% RSLogix 500 project P2_BAK007.RSS, saved by version 8.30.00.16 %
PROJECT "UNTITLED"    % processor: Bul.1763 MicroLogix 1100 Series B %

PROGRAM FILES
  LAD 2 "MAIN"  4 rungs
  LAD 3 "I/O"  8 rungs
  LAD 4 "CONTROLS"  6 rungs
  LAD 5 "CYCLE"  5 rungs

DATA FILES
  O0 OUTPUT  4 elements
  I1 INPUT  6 elements
  S2 STATUS  66 elements
  B3 BINARY  6 elements
  T4 TIMER  1 elements
  C5 COUNTER  1 elements
  R6 CONTROL  1 elements
  N7 INTEGER  1 elements
  F8 FLOAT  1 elements

LADDER 2 "MAIN"
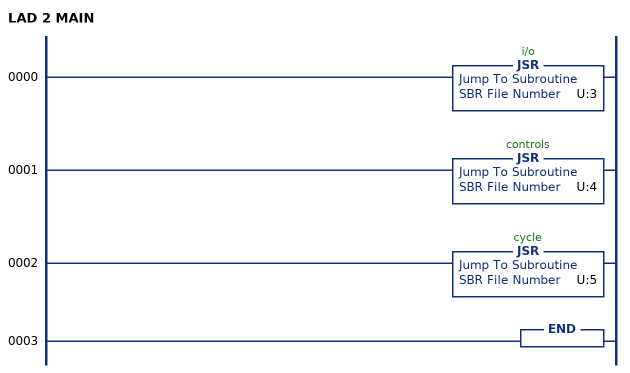
% Rung: 0 %
SOR JSR U:3 EOR
%   U:3  "i/o" %
% Rung: 1 %
SOR JSR U:4 EOR
%   U:4  "controls" %
% Rung: 2 %
SOR JSR U:5 EOR
%   U:5  "cycle" %
% Rung: 3 %
SOR END EOR

LADDER 3 "I/O"
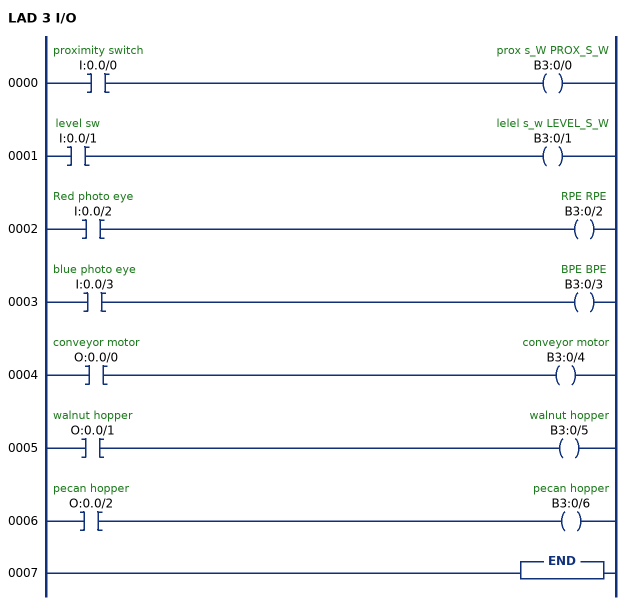
% Rung: 0 %
SOR XIC I:0.0/0 OTE B3:0/0 EOR
%   I:0.0/0  "proximity switch" %
%   B3:0/0  PROX_S_W  "prox s_W" %
% Rung: 1 %
SOR XIC I:0.0/1 OTE B3:0/1 EOR
%   I:0.0/1  "level sw" %
%   B3:0/1  LEVEL_S_W  "lelel s_w" %
% Rung: 2 %
SOR XIC I:0.0/2 OTE B3:0/2 EOR
%   I:0.0/2  "Red photo eye" %
%   B3:0/2  RPE  "RPE" %
% Rung: 3 %
SOR XIC I:0.0/3 OTE B3:0/3 EOR
%   I:0.0/3  "blue photo eye" %
%   B3:0/3  BPE  "BPE" %
% Rung: 4 %
SOR XIC O:0.0/0 OTE B3:0/4 EOR
%   O:0.0/0  "conveyor motor" %
%   B3:0/4  "conveyor motor" %
% Rung: 5 %
SOR XIC O:0.0/1 OTE B3:0/5 EOR
%   O:0.0/1  "walnut hopper" %
%   B3:0/5  "walnut hopper" %
% Rung: 6 %
SOR XIC O:0.0/2 OTE B3:0/6 EOR
%   O:0.0/2  "pecan hopper" %
%   B3:0/6  "pecan hopper" %
% Rung: 7 %
SOR END EOR

LADDER 4 "CONTROLS"
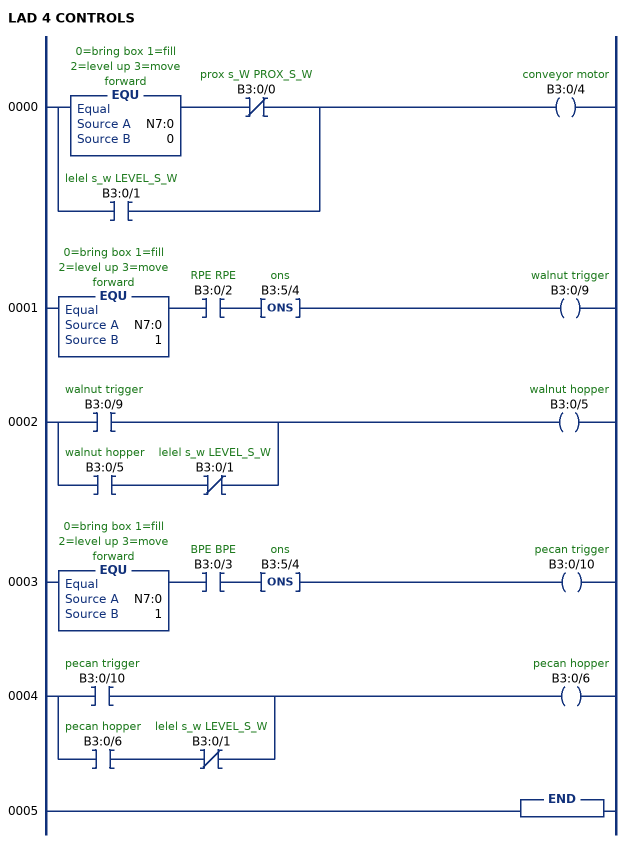
% Rung: 0 %
SOR BST EQU N7:0 0 XIO B3:0/0 NXB XIC B3:0/1 BND OTE B3:0/4 EOR
%   N7:0  "0=bring box 1=fill 2=level up 3=move forward" %
%   B3:0/0  PROX_S_W  "prox s_W" %
%   B3:0/1  LEVEL_S_W  "lelel s_w" %
%   B3:0/4  "conveyor motor" %
% Rung: 1 %
SOR EQU N7:0 1 XIC B3:0/2 ONS B3:5/4 OTE B3:0/9 EOR
%   N7:0  "0=bring box 1=fill 2=level up 3=move forward" %
%   B3:0/2  RPE  "RPE" %
%   B3:5/4  "ons" %
%   B3:0/9  "walnut trigger" %
% Rung: 2 %
SOR BST XIC B3:0/9 NXB XIC B3:0/5 XIO B3:0/1 BND OTE B3:0/5 EOR
%   B3:0/9  "walnut trigger" %
%   B3:0/5  "walnut hopper" %
%   B3:0/1  LEVEL_S_W  "lelel s_w" %
% Rung: 3 %
SOR EQU N7:0 1 XIC B3:0/3 ONS B3:5/4 OTE B3:0/10 EOR
%   N7:0  "0=bring box 1=fill 2=level up 3=move forward" %
%   B3:0/3  BPE  "BPE" %
%   B3:5/4  "ons" %
%   B3:0/10  "pecan trigger" %
% Rung: 4 %
SOR BST XIC B3:0/10 NXB XIC B3:0/6 XIO B3:0/1 BND OTE B3:0/6 EOR
%   B3:0/10  "pecan trigger" %
%   B3:0/6  "pecan hopper" %
%   B3:0/1  LEVEL_S_W  "lelel s_w" %
% Rung: 5 %
SOR END EOR

LADDER 5 "CYCLE"
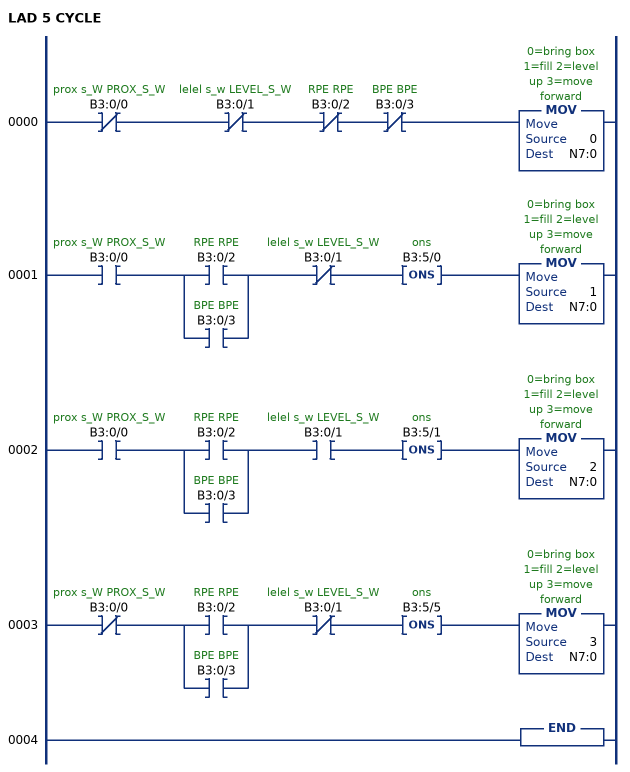
% Rung: 0 %
SOR XIO B3:0/0 XIO B3:0/1 XIO B3:0/2 XIO B3:0/3 MOV 0 N7:0 EOR
%   B3:0/0  PROX_S_W  "prox s_W" %
%   B3:0/1  LEVEL_S_W  "lelel s_w" %
%   B3:0/2  RPE  "RPE" %
%   B3:0/3  BPE  "BPE" %
%   N7:0  "0=bring box 1=fill 2=level up 3=move forward" %
% Rung: 1 %
SOR XIC B3:0/0 BST XIC B3:0/2 NXB XIC B3:0/3 BND XIO B3:0/1 ONS B3:5/0 MOV 1 N7:0 EOR
%   B3:0/0  PROX_S_W  "prox s_W" %
%   B3:0/2  RPE  "RPE" %
%   B3:0/3  BPE  "BPE" %
%   B3:0/1  LEVEL_S_W  "lelel s_w" %
%   B3:5/0  "ons" %
%   N7:0  "0=bring box 1=fill 2=level up 3=move forward" %
% Rung: 2 %
SOR XIC B3:0/0 BST XIC B3:0/2 NXB XIC B3:0/3 BND XIC B3:0/1 ONS B3:5/1 MOV 2 N7:0 EOR
%   B3:0/0  PROX_S_W  "prox s_W" %
%   B3:0/2  RPE  "RPE" %
%   B3:0/3  BPE  "BPE" %
%   B3:0/1  LEVEL_S_W  "lelel s_w" %
%   B3:5/1  "ons" %
%   N7:0  "0=bring box 1=fill 2=level up 3=move forward" %
% Rung: 3 %
SOR XIO B3:0/0 BST XIC B3:0/2 NXB XIC B3:0/3 BND XIO B3:0/1 ONS B3:5/5 MOV 3 N7:0 EOR
%   B3:0/0  PROX_S_W  "prox s_W" %
%   B3:0/2  RPE  "RPE" %
%   B3:0/3  BPE  "BPE" %
%   B3:0/1  LEVEL_S_W  "lelel s_w" %
%   B3:5/5  "ons" %
%   N7:0  "0=bring box 1=fill 2=level up 3=move forward" %
% Rung: 4 %
SOR END EOR

OTHER DOCUMENTED ADDRESSES
  B3:0/7  "conveyor trigger"
  B3:0/8  "conveyor interupt"
  B3:2/0  "ebit"
  B3:3/0  "trigger"
  B3:3/1  "trigger"
  B3:4/0  "ons"
  B3:5/3  "ons"
  B4:4/0  "ons"
  N7:1  "bring box =0 fill mod=1 level up=2"
  ONS  "one shot"
